FUNCTION_BLOCK FB_ControllerBase_SFC
VAR CONSTANT
	MAX_ERRORS	: UINT := 10;
	MAX_TIMEOUT	: TIME := T#30S;
END_VAR
VAR_INPUT
	dr			: REFERENCE TO FB_Director;	
	IC			: BOOL;
	Execute		: BOOL;
	Ack			: BOOL;	
	SFCPause	: BOOL;
	SFCReset	: BOOL;
	UnsafeStop 	: BOOL := FALSE;
	Clocks		: ARRAY[1..MAX_ERRORS]	OF TON; // max_errors
END_VAR
VAR_OUTPUT
	Ready		: BOOL;
	//Failure		: BOOL;
	NumError	: UINT := 0;
	Done		: BOOL := FALSE;
	Timed		: ARRAY[1..MAX_ERRORS]	OF BOOL; // 
	//RTrigs		: ARRAY[1..MAX_ERRORS]	OF R_TRIG;
	//Timeouts	: ARRAY[1...MAX_ERRORS]	OF TIME;
END_VAR

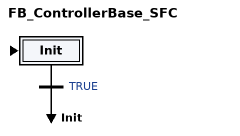
INITIAL_STEP Init:
END_STEP
TRANSITION FROM Init TO Init
    := TRUE;
END_TRANSITION

METHOD FB_init : BOOL
VAR_INPUT
	bInitRetains : BOOL; // if TRUE, the retain variables are initialized (warm start / cold start)
	bInCopyCode : BOOL;  // if TRUE, the instance afterwards gets moved into the copy code (online change)
END_VAR

VAR 
	I: UINT;
END_VAR
FOR I:=1 TO MAX_ERRORS DO
	Timed[i] 		:= FALSE;
	//RTrigs[i].CLK 	:= Timed[i];
	// Timeouts[I] 	:= MAX_TIMEOUT;
	Clocks[i].IN	:= Timed[i]; // := MAX_TIMEOUT;
	Clocks[i].PT	:= MAX_TIMEOUT;
	//RTrigs[i].CLK	:= FALSE;
	//Clocks[i].Q
END_FOR
END_METHOD

METHOD IsPaused : BOOL
IsPaused := SFCPause;
END_METHOD

METHOD PauseAndReset : BOOL
VAR_INPUT
	gmModeActual 	: E_GEMMA;
END_VAR
VAR 
	fp : R_TRIG;
	i : UINT;
END_VAR
fp(CLK:=(gmModeActual = E_GEMMA.A6Inicializando), Q=> SFCReset);
SFCPause := NOT UnsafeStop AND (NumError <> 0 OR gmModeActual=E_GEMMA.A3ParadaEstado OR gmModeActual=E_GEMMA.A4ParadaObtenida or gmModeActual=E_GEMMA.D2TratamientoFallos);

//Clocks[1](IN:= Timed[1], PT:=T#5S);

//Clocks[1].PT := t#5s; // MAX_TIMEOUT;
FOR i:= 1 TO MAX_ERRORS DO
	//Clocks[i].PT := MAX_TIMEOUT;
//	Clocks[i].IN := Timed[i];
	//IF Timed[i] THEN
		 // := TRUE;
		
	Clocks[i](IN:= Timed[i], PT:=MAX_TIMEOUT);
	//RTrigs[I].CLK:=  Timed[i];
	//IF RTrigs[I].Q THEN 
	//Clocks[i].IN := TRUE;
	//ELSIF NOT Timed[I] THEN
	//ELSE
		//Clocks[I].IN := FALSE;
	// END_IF
	IF Clocks[i].Q THEN
		NumError := i;
	END_IF
END_FOR
//*)
END_METHOD

END_FUNCTION_BLOCK

(* stored: Version 1.1.0.1, ProductVersion 3.1.4024.11
   POU FB_ControllerBase_SFC: Id {b4a568e5-b860-4b97-ba61-d1f48d9d8c8d}, SpecialFunc None
   Method FB_init: Id {0d874f96-f55f-4d86-871c-77c076024b66}
   Method IsPaused: Id {e98f7813-c900-4fd4-9a12-006983f9c884}
   Method PauseAndReset: Id {c358a4ee-9530-49d3-9f5f-b83d275d2af8} *)
